INTERFACE I_LightTower

// Provides access to buzzer control
PROPERTY Buzzer : I_LightTowerComponent
GET
END_GET
END_PROPERTY

// Provides access to green light control
PROPERTY GreenLight : I_LightTowerComponent
GET
END_GET
END_PROPERTY

// Provides access to orange light control
PROPERTY OrangeLight : I_LightTowerComponent
GET
END_GET
END_PROPERTY

// Provides access to red light control
PROPERTY RedLight : I_LightTowerComponent
GET
END_GET
END_PROPERTY

END_INTERFACE

(* stored: Version 1.1.0.1, ProductVersion 3.1.4024.14
   Itf I_LightTower: Id {d87fa2f2-d844-0bb2-2300-f6f03f34bfc0}
   Property Buzzer: Id {772d8f2c-e516-05be-3194-96f6b72a7410}
   Get Get: Id {68936fea-43c9-024f-0f21-30e47ad6f507}
   Property GreenLight: Id {73752581-7c45-0126-38c6-c3c8f5bcdd08}
   Get Get: Id {1e68cb49-791e-0f38-2aa7-0f4b99164dfa}
   Property OrangeLight: Id {fb0decf6-5d47-05d9-199f-fb2daa1a6f2b}
   Get Get: Id {51c5362f-5f4b-0131-0536-04c9c1c2d11f}
   Property RedLight: Id {39555fe8-b5f7-0a54-00b0-d0aa8d72a53a}
   Get Get: Id {fe772568-97e8-06f1-0425-ec3df04f54c2} *)
